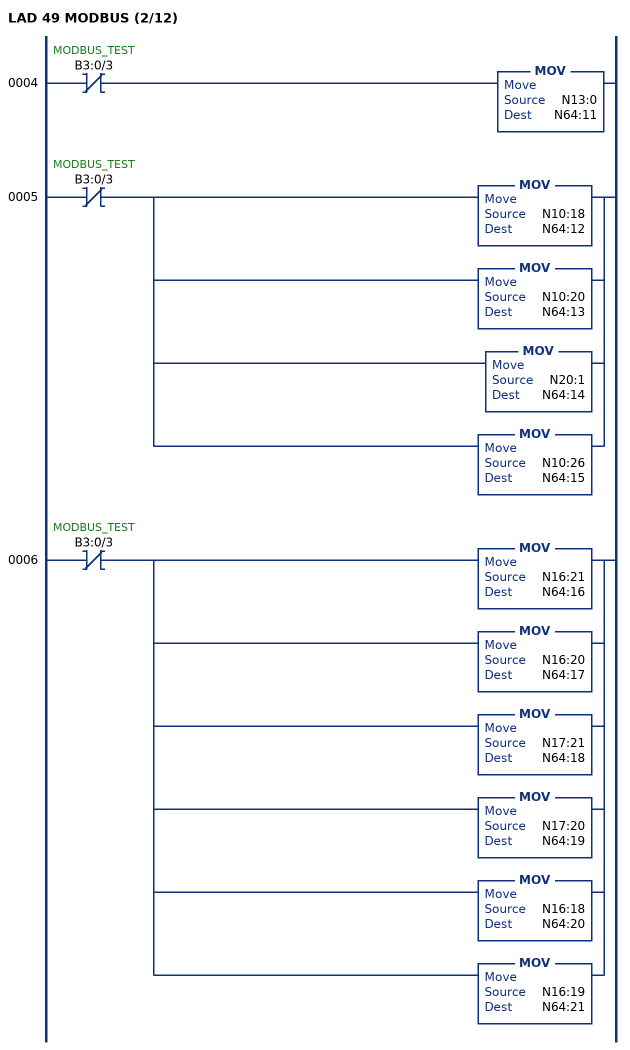
% Rung: 4 %
SOR XIO B3:0/3 MOV N13:0 N64:11 EOR
%   B3:0/3  MODBUS_TEST %
%   N13:0  REGEN_STATE  "STATE The current state of the regen process" %
% Rung: 5 %
SOR XIO B3:0/3 BST MOV N10:18 N64:12 NXB MOV N10:20 N64:13 NXB MOV N20:1 N64:14 NXB MOV N10:26 N64:15 BND EOR
%   B3:0/3  MODBUS_TEST %
%   N10:18  INLET_PX_PSIG %
%   N10:20  OUTLET_PX_PSIG %
%   N20:1  MIX_PANEL_PSIG %
%   N10:26  MFM_FLOW %
% Rung: 6 %
SOR XIO B3:0/3 BST MOV N16:21 N64:16 NXB MOV N16:20 N64:17 NXB MOV N17:21 N64:18 NXB MOV N17:20 N64:19 NXB MOV N16:18 N64:20 NXB MOV N16:19 N64:21 BND EOR
%   B3:0/3  MODBUS_TEST %
%   N16:21  ADS_A_BED_TEMP_READ %
%   N16:20  ADS_A_WALL_TEMP_READ %
%   N17:21  ADS_B_BED_TEMP_READ %
%   N17:20  ADS_B_WALL_TEMP_READ %
%   N16:18  ADS_PH_GAS_TEMP_READ %
%   N16:19  ADS_PH_ROD_TEMP_READ %

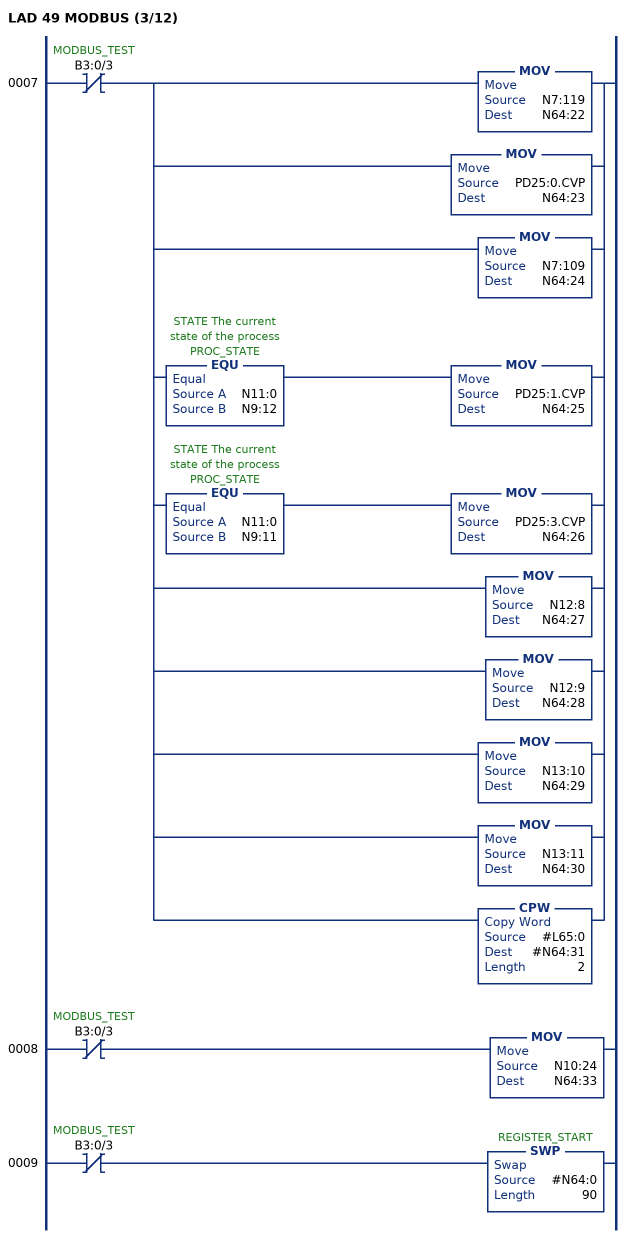
% Rung: 7 %
SOR XIO B3:0/3 BST MOV N7:119 N64:22 NXB MOV PD25:0.CVP N64:23 NXB MOV N7:109 N64:24 NXB EQU N11:0 N9:12 MOV PD25:1.CVP N64:25 NXB EQU N11:0 N9:11 MOV PD25:3.CVP N64:26 NXB MOV N12:8 N64:27 NXB MOV N12:9 N64:28 NXB MOV N13:10 N64:29 NXB MOV N13:11 N64:30 NXB CPW #L65:0 #N64:31 2 BND EOR
%   B3:0/3  MODBUS_TEST %
%   N7:119  PREHEATER_SP  "CONTROL Preheater PID Setpoint" %
%   N7:109  BLANKET_SP  "CONTROL Blanket PID Setpoint" %
%   N11:0  PROC_STATE  "STATE The current state of the process" %
%   N9:12  PROC_PURIFY_B  "STATE Process Purify B" %
%   N9:11  PROC_PURIFY_A  "STATE Process Purify A" %
%   N12:8  HRS_LEFT_IN_PURIFY %
%   N12:9  MIN_LEFT_IN_PURIFY %
%   N13:10  REGEN_HRS_LEFT  "STATUS Regen Preheater Temperature Initial Temperature" %
%   N13:11  REGEN_MIN_LEFT  "STATUS Preheater Alarm Measured temperature change" %
%   L65:0  TOTAL_FLOW %
% Rung: 8 %
SOR XIO B3:0/3 MOV N10:24 N64:33 EOR
%   B3:0/3  MODBUS_TEST %
%   N10:24  H2_SENSOR_LEVEL %
% Rung: 9 %
SOR XIO B3:0/3 SWP #N64:0 90 EOR
%   B3:0/3  MODBUS_TEST %
%   N64:0  REGISTER_START %

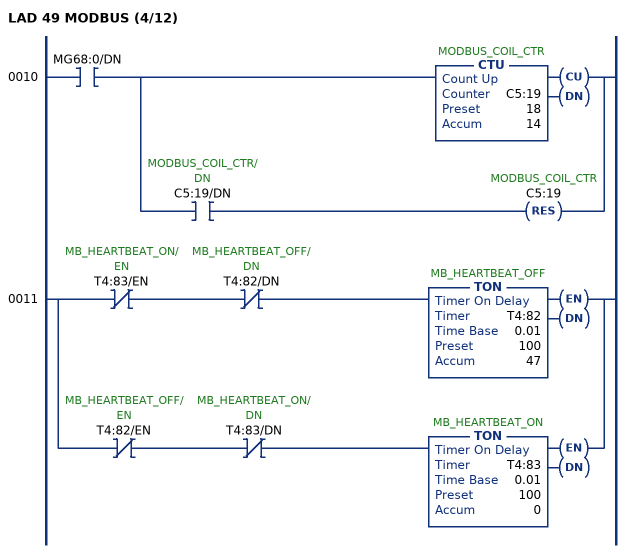
% Rung: 10 %
SOR XIC MG68:0/DN BST CTU C5:19 18 14 NXB XIC C5:19/DN RES C5:19 BND EOR
%   C5:19  MODBUS_COIL_CTR %
% Rung: 11 %
SOR BST XIO T4:83/EN XIO T4:82/DN TON T4:82 0.01 100 47 NXB XIO T4:82/EN XIO T4:83/DN TON T4:83 0.01 100 0 BND EOR
%   T4:83  MB_HEARTBEAT_ON %
%   T4:82  MB_HEARTBEAT_OFF %

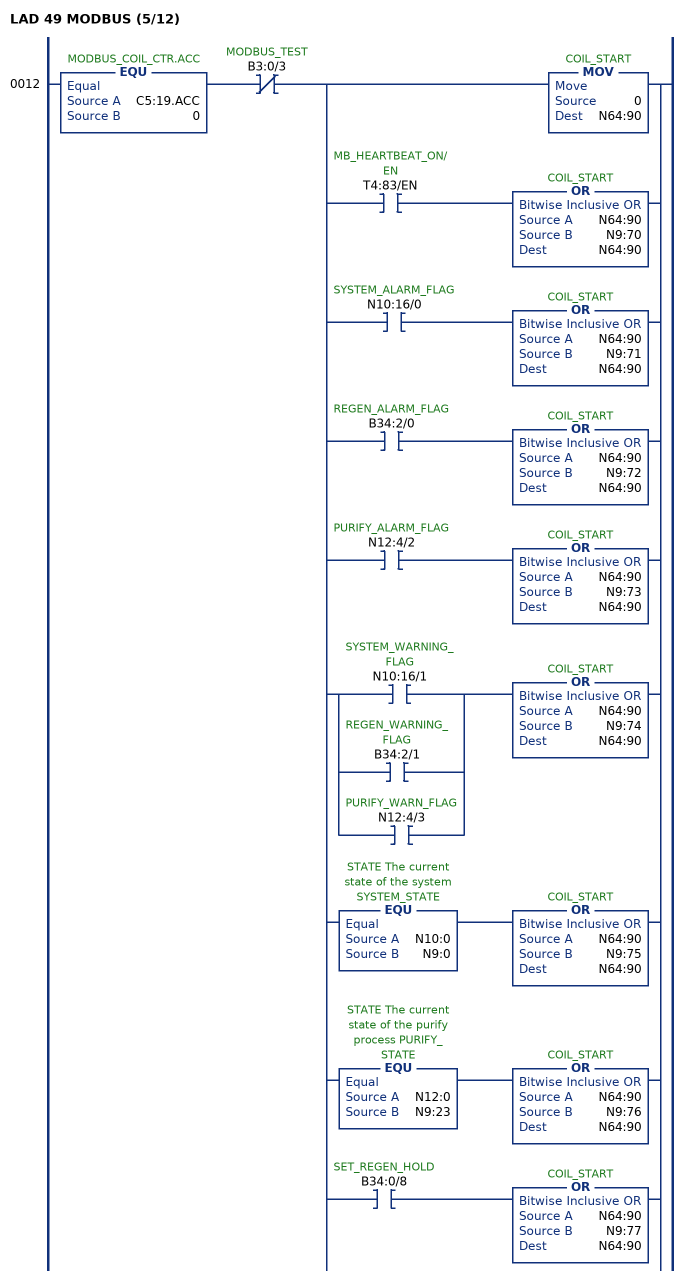

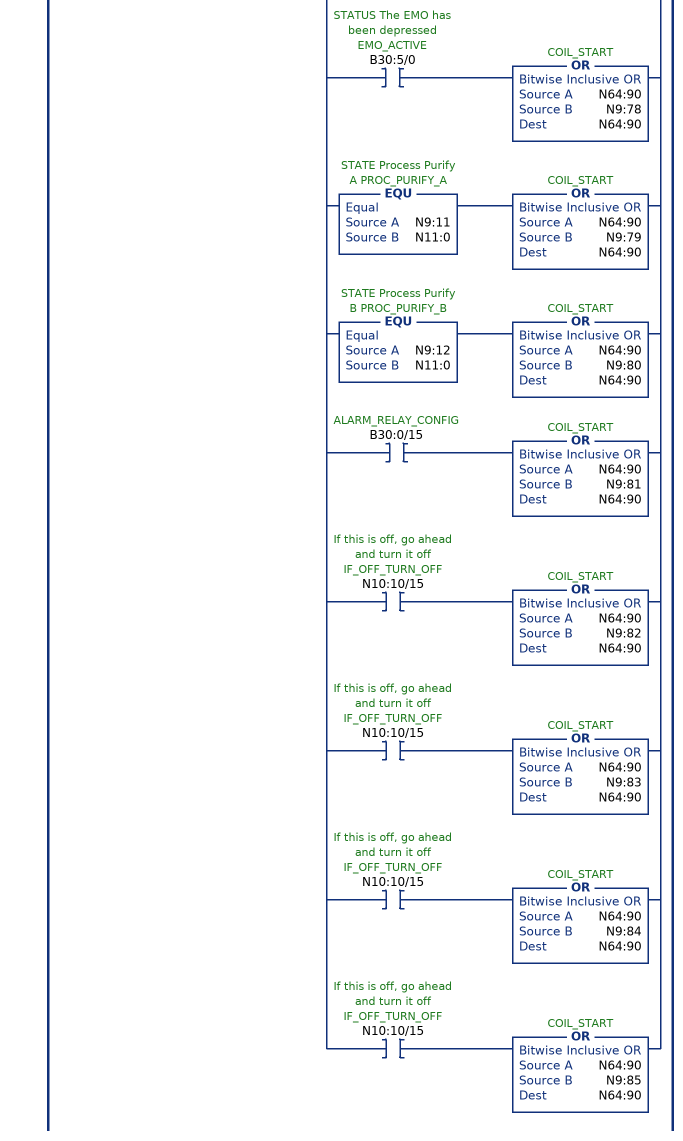
% Rung: 12 %
SOR EQU C5:19.ACC 0 XIO B3:0/3 BST MOV 0 N64:90 NXB XIC T4:83/EN OR N64:90 N9:70 N64:90 NXB XIC N10:16/0 OR N64:90 N9:71 N64:90 NXB XIC B34:2/0 OR N64:90 N9:72 N64:90 NXB XIC N12:4/2 OR N64:90 N9:73 N64:90 NXB BST XIC N10:16/1 NXB XIC B34:2/1 NXB XIC N12:4/3 BND OR N64:90 N9:74 N64:90 NXB EQU N10:0 N9:0 OR N64:90 N9:75 N64:90 NXB EQU N12:0 N9:23 OR N64:90 N9:76 N64:90 NXB XIC B34:0/8 OR N64:90 N9:77 N64:90 NXB XIC B30:5/0 OR N64:90 N9:78 N64:90 NXB EQU N9:11 N11:0 OR N64:90 N9:79 N64:90 NXB EQU N9:12 N11:0 OR N64:90 N9:80 N64:90 NXB XIC B30:0/15 OR N64:90 N9:81 N64:90 NXB XIC N10:10/15 OR N64:90 N9:82 N64:90 NXB XIC N10:10/15 OR N64:90 N9:83 N64:90 NXB XIC N10:10/15 OR N64:90 N9:84 N64:90 NXB XIC N10:10/15 OR N64:90 N9:85 N64:90 BND EOR
%   C5:19  MODBUS_COIL_CTR %
%   B3:0/3  MODBUS_TEST %
%   N64:90  COIL_START %
%   T4:83  MB_HEARTBEAT_ON %
%   N9:70  BIT_0 %
%   N10:16/0  SYSTEM_ALARM_FLAG %
%   N9:71  BIT_1 %
%   B34:2/0  REGEN_ALARM_FLAG %
%   N9:72  BIT_2 %
%   N12:4/2  PURIFY_ALARM_FLAG %
%   N9:73  BIT_3 %
%   N10:16/1  SYSTEM_WARNING_FLAG %
%   B34:2/1  REGEN_WARNING_FLAG %
%   N12:4/3  PURIFY_WARN_FLAG %
%   N9:74  BIT_4 %
%   N10:0  SYSTEM_STATE  "STATE The current state of the system" %
%   N9:0  SYSTEM_STANDBY  "STATE System Standby" %
%   N9:75  BIT_5 %
%   N12:0  PURIFY_STATE  "STATE The current state of the purify process" %
%   N9:23  PURIFY_MANUAL_HOLD  "STATE Purify Manual Hold" %
%   N9:76  BIT_6 %
%   B34:0/8  SET_REGEN_HOLD %
%   N9:77  BIT_7 %
%   B30:5/0  EMO_ACTIVE  "STATUS The EMO has been depressed" %
%   N9:78  BIT_8 %
%   N9:11  PROC_PURIFY_A  "STATE Process Purify A" %
%   N11:0  PROC_STATE  "STATE The current state of the process" %
%   N9:79  BIT_9 %
%   N9:12  PROC_PURIFY_B  "STATE Process Purify B" %
%   N9:80  BIT_10 %
%   B30:0/15  ALARM_RELAY_CONFIG %
%   N9:81  BIT_11 %
%   N10:10/15  IF_OFF_TURN_OFF  "If this is off, go ahead and turn it off" %
%   N9:82  BIT_12 %
%   N9:83  BIT_13 %
%   N9:84  BIT_14 %
%   N9:85  BIT_15 %

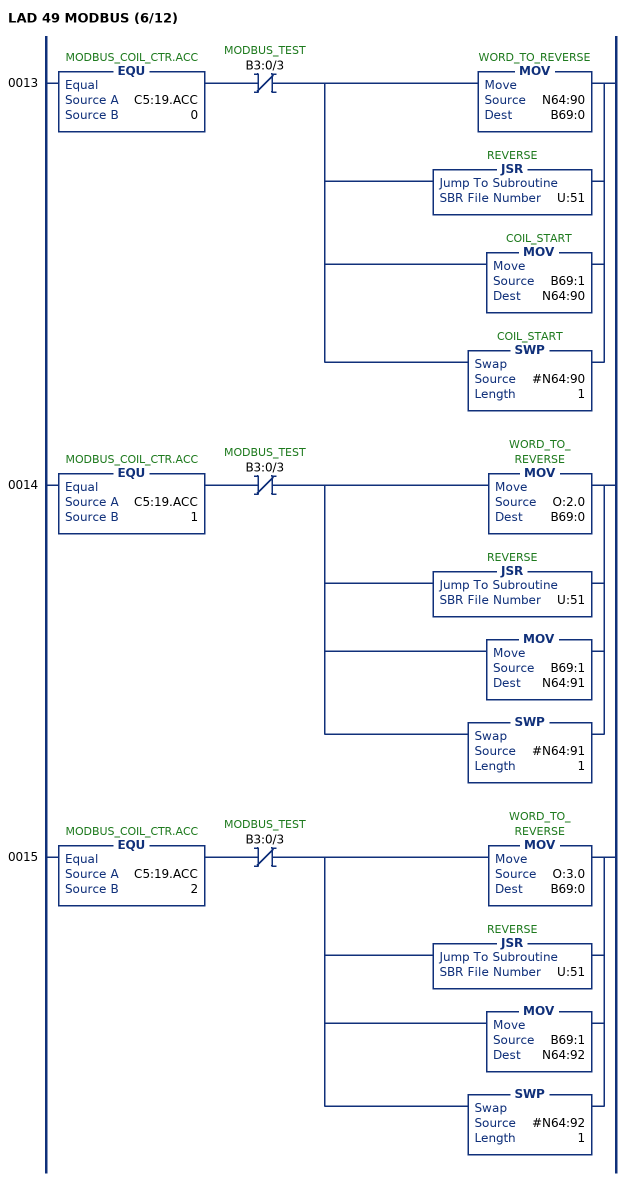
% Rung: 13 %
SOR EQU C5:19.ACC 0 XIO B3:0/3 BST MOV N64:90 B69:0 NXB JSR U:51 NXB MOV B69:1 N64:90 NXB SWP #N64:90 1 BND EOR
%   C5:19  MODBUS_COIL_CTR %
%   B3:0/3  MODBUS_TEST %
%   N64:90  COIL_START %
%   B69:0  WORD_TO_REVERSE %
%   U:51  REVERSE %
%   B69:1  REVERSED_WORD %
% Rung: 14 %
SOR EQU C5:19.ACC 1 XIO B3:0/3 BST MOV O:2.0 B69:0 NXB JSR U:51 NXB MOV B69:1 N64:91 NXB SWP #N64:91 1 BND EOR
%   C5:19  MODBUS_COIL_CTR %
%   B3:0/3  MODBUS_TEST %
%   B69:0  WORD_TO_REVERSE %
%   U:51  REVERSE %
%   B69:1  REVERSED_WORD %
% Rung: 15 %
SOR EQU C5:19.ACC 2 XIO B3:0/3 BST MOV O:3.0 B69:0 NXB JSR U:51 NXB MOV B69:1 N64:92 NXB SWP #N64:92 1 BND EOR
%   C5:19  MODBUS_COIL_CTR %
%   B3:0/3  MODBUS_TEST %
%   B69:0  WORD_TO_REVERSE %
%   U:51  REVERSE %
%   B69:1  REVERSED_WORD %

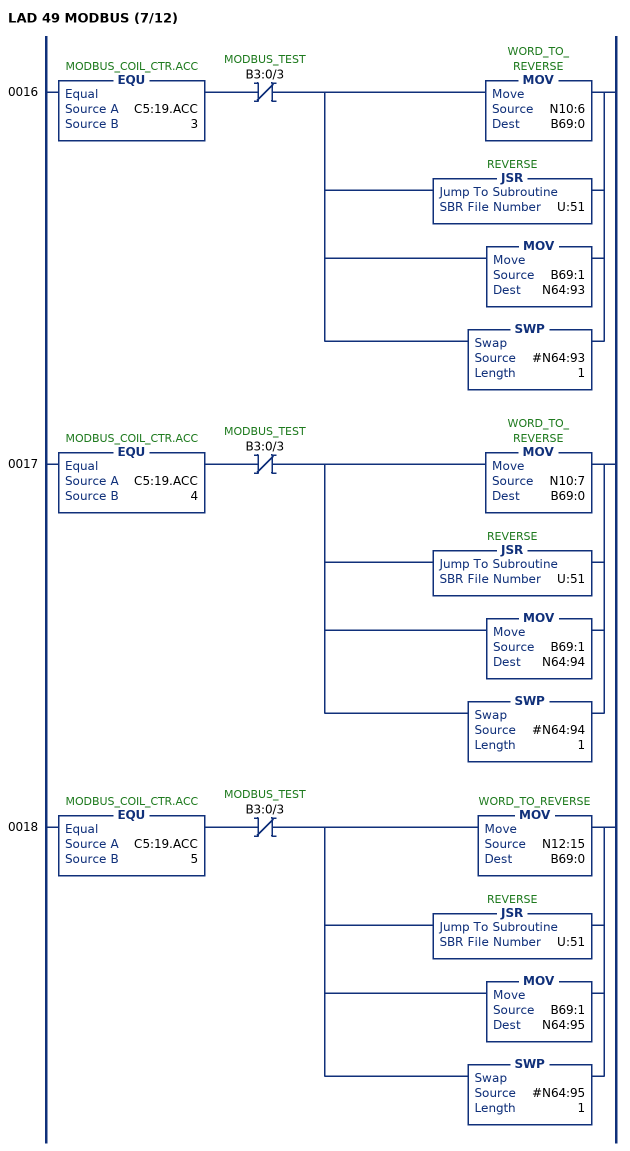
% Rung: 16 %
SOR EQU C5:19.ACC 3 XIO B3:0/3 BST MOV N10:6 B69:0 NXB JSR U:51 NXB MOV B69:1 N64:93 NXB SWP #N64:93 1 BND EOR
%   C5:19  MODBUS_COIL_CTR %
%   B3:0/3  MODBUS_TEST %
%   N10:6  SYSTEM_ALARMS_0  "ALARM System alarms" %
%   B69:0  WORD_TO_REVERSE %
%   U:51  REVERSE %
%   B69:1  REVERSED_WORD %
% Rung: 17 %
SOR EQU C5:19.ACC 4 XIO B3:0/3 BST MOV N10:7 B69:0 NXB JSR U:51 NXB MOV B69:1 N64:94 NXB SWP #N64:94 1 BND EOR
%   C5:19  MODBUS_COIL_CTR %
%   B3:0/3  MODBUS_TEST %
%   N10:7  SYSTEM_ALARMS_1  "ALARM System alarms" %
%   B69:0  WORD_TO_REVERSE %
%   U:51  REVERSE %
%   B69:1  REVERSED_WORD %
% Rung: 18 %
SOR EQU C5:19.ACC 5 XIO B3:0/3 BST MOV N12:15 B69:0 NXB JSR U:51 NXB MOV B69:1 N64:95 NXB SWP #N64:95 1 BND EOR
%   C5:19  MODBUS_COIL_CTR %
%   B3:0/3  MODBUS_TEST %
%   N12:15  PURIFY_ALARMS_0 %
%   B69:0  WORD_TO_REVERSE %
%   U:51  REVERSE %
%   B69:1  REVERSED_WORD %

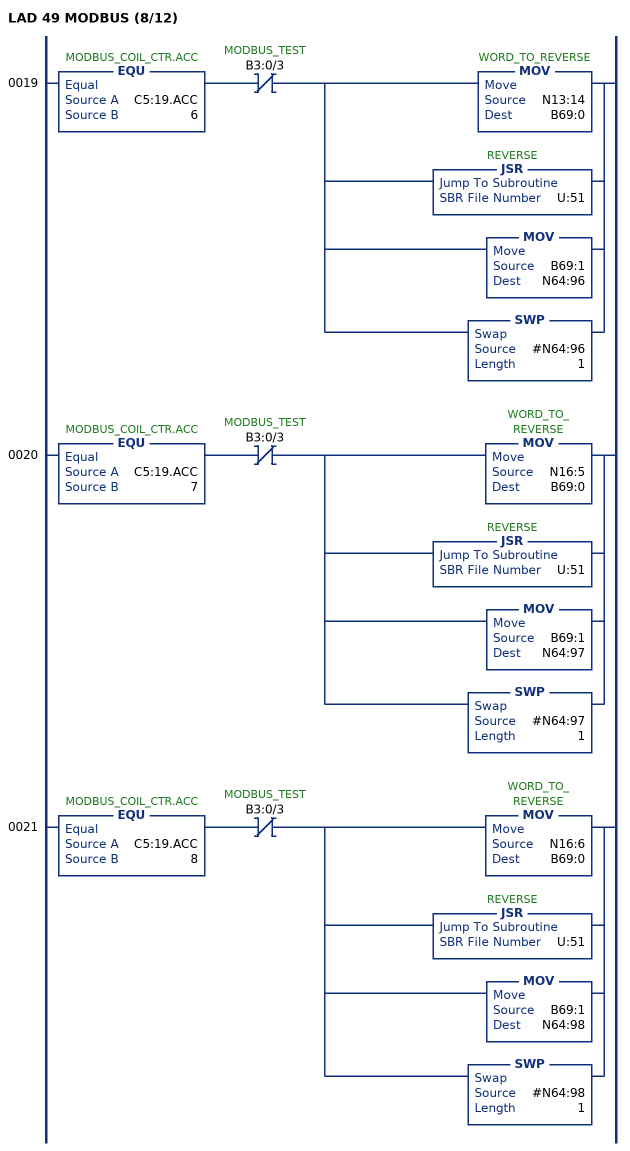
% Rung: 19 %
SOR EQU C5:19.ACC 6 XIO B3:0/3 BST MOV N13:14 B69:0 NXB JSR U:51 NXB MOV B69:1 N64:96 NXB SWP #N64:96 1 BND EOR
%   C5:19  MODBUS_COIL_CTR %
%   B3:0/3  MODBUS_TEST %
%   N13:14  REGEN_ALARMS_0 %
%   B69:0  WORD_TO_REVERSE %
%   U:51  REVERSE %
%   B69:1  REVERSED_WORD %
% Rung: 20 %
SOR EQU C5:19.ACC 7 XIO B3:0/3 BST MOV N16:5 B69:0 NXB JSR U:51 NXB MOV B69:1 N64:97 NXB SWP #N64:97 1 BND EOR
%   C5:19  MODBUS_COIL_CTR %
%   B3:0/3  MODBUS_TEST %
%   N16:5  ADS_A_ALARMS_0  "ALARM ADS A Alarms" %
%   B69:0  WORD_TO_REVERSE %
%   U:51  REVERSE %
%   B69:1  REVERSED_WORD %
% Rung: 21 %
SOR EQU C5:19.ACC 8 XIO B3:0/3 BST MOV N16:6 B69:0 NXB JSR U:51 NXB MOV B69:1 N64:98 NXB SWP #N64:98 1 BND EOR
%   C5:19  MODBUS_COIL_CTR %
%   B3:0/3  MODBUS_TEST %
%   N16:6  ADS_A_ALARMS_1  "ALARM ADS A Alarms" %
%   B69:0  WORD_TO_REVERSE %
%   U:51  REVERSE %
%   B69:1  REVERSED_WORD %

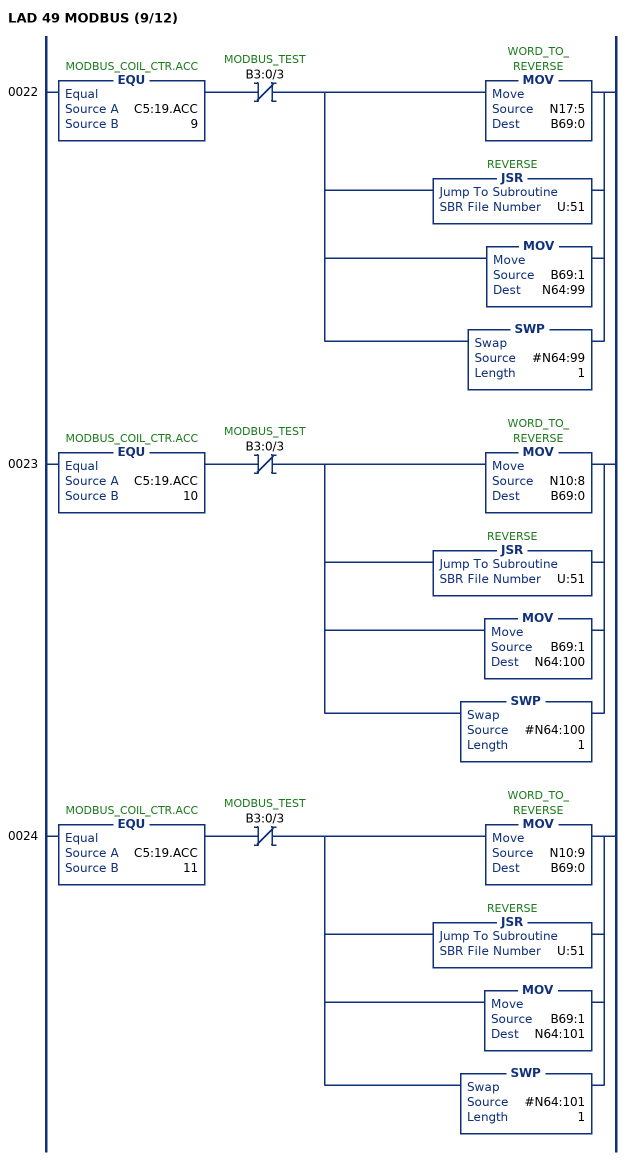
% Rung: 22 %
SOR EQU C5:19.ACC 9 XIO B3:0/3 BST MOV N17:5 B69:0 NXB JSR U:51 NXB MOV B69:1 N64:99 NXB SWP #N64:99 1 BND EOR
%   C5:19  MODBUS_COIL_CTR %
%   B3:0/3  MODBUS_TEST %
%   N17:5  ADS_B_ALARMS_0  "ALARM Alarm bits" %
%   B69:0  WORD_TO_REVERSE %
%   U:51  REVERSE %
%   B69:1  REVERSED_WORD %
% Rung: 23 %
SOR EQU C5:19.ACC 10 XIO B3:0/3 BST MOV N10:8 B69:0 NXB JSR U:51 NXB MOV B69:1 N64:100 NXB SWP #N64:100 1 BND EOR
%   C5:19  MODBUS_COIL_CTR %
%   B3:0/3  MODBUS_TEST %
%   N10:8  SYSTEM_WARNINGS_0  "WARNING System Warnings" %
%   B69:0  WORD_TO_REVERSE %
%   U:51  REVERSE %
%   B69:1  REVERSED_WORD %
% Rung: 24 %
SOR EQU C5:19.ACC 11 XIO B3:0/3 BST MOV N10:9 B69:0 NXB JSR U:51 NXB MOV B69:1 N64:101 NXB SWP #N64:101 1 BND EOR
%   C5:19  MODBUS_COIL_CTR %
%   B3:0/3  MODBUS_TEST %
%   N10:9  SYSTEM_WARNINGS_1  "WARNING System Warnings" %
%   B69:0  WORD_TO_REVERSE %
%   U:51  REVERSE %
%   B69:1  REVERSED_WORD %

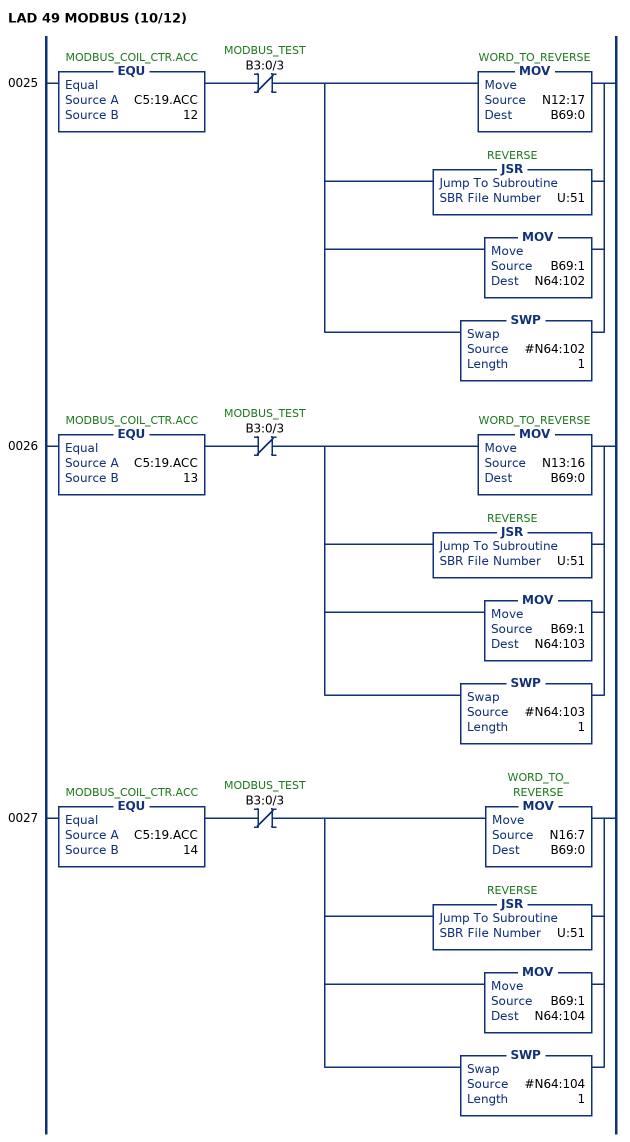
% Rung: 25 %
SOR EQU C5:19.ACC 12 XIO B3:0/3 BST MOV N12:17 B69:0 NXB JSR U:51 NXB MOV B69:1 N64:102 NXB SWP #N64:102 1 BND EOR
%   C5:19  MODBUS_COIL_CTR %
%   B3:0/3  MODBUS_TEST %
%   N12:17  PURIFY_WARNINGS_0 %
%   B69:0  WORD_TO_REVERSE %
%   U:51  REVERSE %
%   B69:1  REVERSED_WORD %
% Rung: 26 %
SOR EQU C5:19.ACC 13 XIO B3:0/3 BST MOV N13:16 B69:0 NXB JSR U:51 NXB MOV B69:1 N64:103 NXB SWP #N64:103 1 BND EOR
%   C5:19  MODBUS_COIL_CTR %
%   B3:0/3  MODBUS_TEST %
%   N13:16  REGEN_WARNINGS_0 %
%   B69:0  WORD_TO_REVERSE %
%   U:51  REVERSE %
%   B69:1  REVERSED_WORD %
% Rung: 27 %
SOR EQU C5:19.ACC 14 XIO B3:0/3 BST MOV N16:7 B69:0 NXB JSR U:51 NXB MOV B69:1 N64:104 NXB SWP #N64:104 1 BND EOR
%   C5:19  MODBUS_COIL_CTR %
%   B3:0/3  MODBUS_TEST %
%   N16:7  ADS_A_WARNINGS_0  "WARNING ADS A Warnings" %
%   B69:0  WORD_TO_REVERSE %
%   U:51  REVERSE %
%   B69:1  REVERSED_WORD %

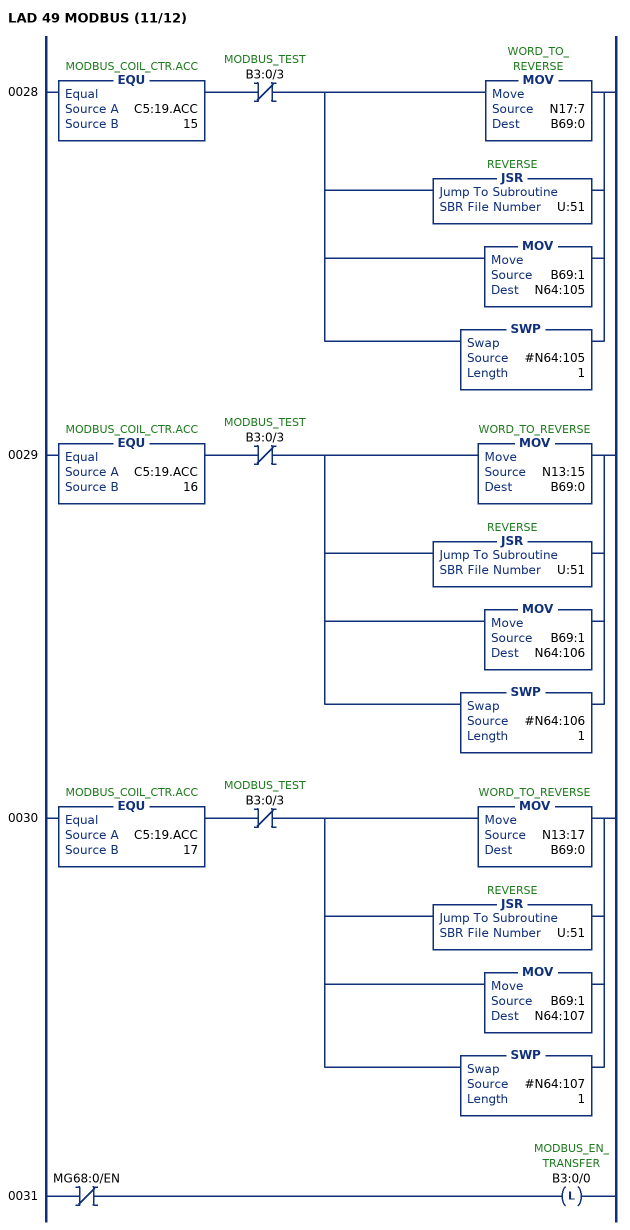
% Rung: 28 %
SOR EQU C5:19.ACC 15 XIO B3:0/3 BST MOV N17:7 B69:0 NXB JSR U:51 NXB MOV B69:1 N64:105 NXB SWP #N64:105 1 BND EOR
%   C5:19  MODBUS_COIL_CTR %
%   B3:0/3  MODBUS_TEST %
%   N17:7  ADS_B_WARNINGS_0  "WARNING Warning bits" %
%   B69:0  WORD_TO_REVERSE %
%   U:51  REVERSE %
%   B69:1  REVERSED_WORD %
% Rung: 29 %
SOR EQU C5:19.ACC 16 XIO B3:0/3 BST MOV N13:15 B69:0 NXB JSR U:51 NXB MOV B69:1 N64:106 NXB SWP #N64:106 1 BND EOR
%   C5:19  MODBUS_COIL_CTR %
%   B3:0/3  MODBUS_TEST %
%   N13:15  REGEN_ALARMS_1 %
%   B69:0  WORD_TO_REVERSE %
%   U:51  REVERSE %
%   B69:1  REVERSED_WORD %
% Rung: 30 %
SOR EQU C5:19.ACC 17 XIO B3:0/3 BST MOV N13:17 B69:0 NXB JSR U:51 NXB MOV B69:1 N64:107 NXB SWP #N64:107 1 BND EOR
%   C5:19  MODBUS_COIL_CTR %
%   B3:0/3  MODBUS_TEST %
%   N13:17  REGEN_WARNINGS_1 %
%   B69:0  WORD_TO_REVERSE %
%   U:51  REVERSE %
%   B69:1  REVERSED_WORD %
% Rung: 31 %
SOR XIO MG68:0/EN OTL B3:0/0 EOR
%   B3:0/0  MODBUS_EN_TRANSFER %

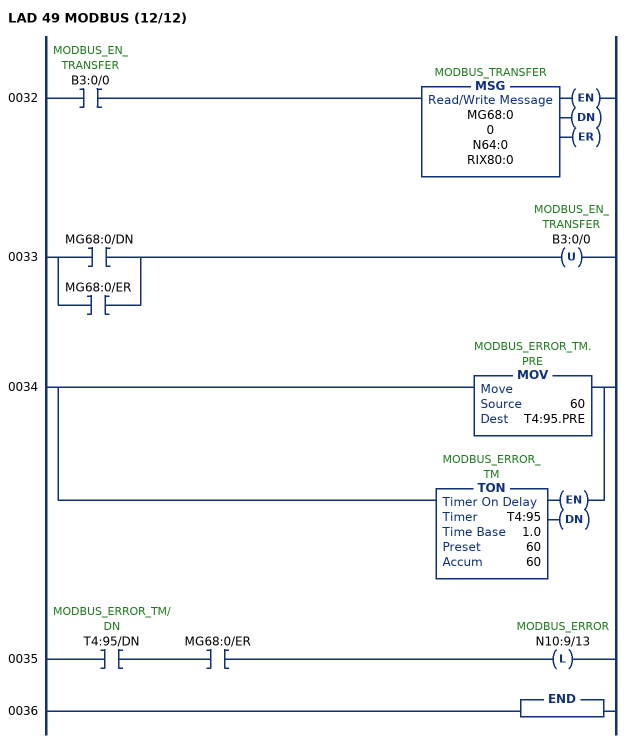
% Rung: 32 %
SOR XIC B3:0/0 MSG MG68:0 0 N64:0 RIX80:0 EOR
%   B3:0/0  MODBUS_EN_TRANSFER %
%   MSG set-up: CIP Generic | 33 | 0 | ? | 0 | 0 | 0 | 0 | 172.16.14.73:502 | 0 | 0 | 172.16.14.73 | RIX80:0 | 10 | 4 | 150 | 3 | 4 | 96 | 3 | 252 | N64:0 %
%   MG68:0  MODBUS_TRANSFER %
%   N64:0  REGISTER_START %
% Rung: 33 %
SOR BST XIC MG68:0/DN NXB XIC MG68:0/ER BND OTU B3:0/0 EOR
%   B3:0/0  MODBUS_EN_TRANSFER %
% Rung: 34 %
SOR BST MOV 60 T4:95.PRE NXB TON T4:95 1.0 60 60 BND EOR
%   T4:95  MODBUS_ERROR_TM %
% Rung: 35 %
SOR XIC T4:95/DN XIC MG68:0/ER OTL N10:9/13 EOR
%   T4:95  MODBUS_ERROR_TM %
%   N10:9/13  MODBUS_ERROR %
% Rung: 36 %
SOR END EOR

LADDER 50 "PLC_FAULT"
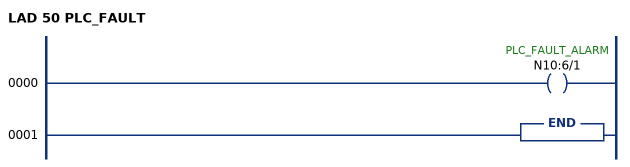
% Rung: 0 %
SOR OTE N10:6/1 EOR
%   N10:6/1  PLC_FAULT_ALARM %
% Rung: 1 %
SOR END EOR

LADDER 51 "REVERSE"
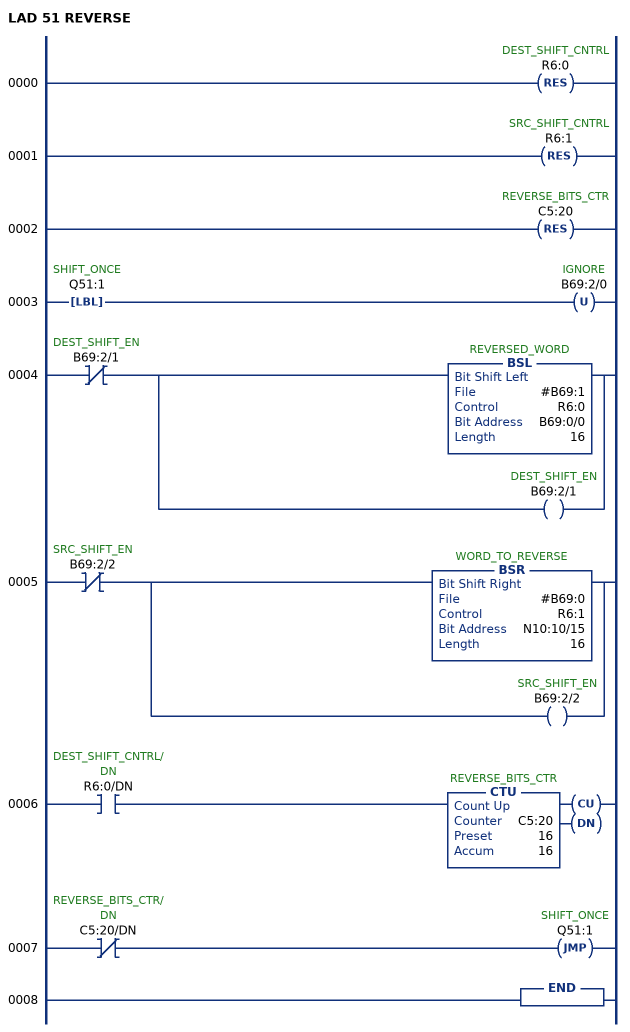
% Rung: 0 %
SOR RES R6:0 EOR
%   R6:0  DEST_SHIFT_CNTRL %
% Rung: 1 %
SOR RES R6:1 EOR
%   R6:1  SRC_SHIFT_CNTRL %
% Rung: 2 %
SOR RES C5:20 EOR
%   C5:20  REVERSE_BITS_CTR %
% Rung: 3 %
SOR LBL Q51:1 OTU B69:2/0 EOR
%   Q51:1  SHIFT_ONCE %
%   B69:2/0  IGNORE %
% Rung: 4 %
SOR XIO B69:2/1 BST BSL #B69:1 R6:0 B69:0/0 16 NXB OTE B69:2/1 BND EOR
%   B69:2/1  DEST_SHIFT_EN %
%   B69:1  REVERSED_WORD %
%   R6:0  DEST_SHIFT_CNTRL %
% Rung: 5 %
SOR XIO B69:2/2 BST BSR #B69:0 R6:1 N10:10/15 16 NXB OTE B69:2/2 BND EOR
%   B69:2/2  SRC_SHIFT_EN %
%   B69:0  WORD_TO_REVERSE %
%   R6:1  SRC_SHIFT_CNTRL %
%   N10:10/15  IF_OFF_TURN_OFF  "If this is off, go ahead and turn it off" %
% Rung: 6 %
SOR XIC R6:0/DN CTU C5:20 16 16 EOR
%   R6:0  DEST_SHIFT_CNTRL %
%   C5:20  REVERSE_BITS_CTR %
% Rung: 7 %
SOR XIO C5:20/DN JMP Q51:1 EOR
%   C5:20  REVERSE_BITS_CTR %
%   Q51:1  SHIFT_ONCE %
% Rung: 8 %
SOR END EOR

OTHER DOCUMENTED ADDRESSES
  B26:2/2  H2_LEAK_ALM_EN
  B30:0  CONFIG_BITS_HARDWARE  "CONFIG Hardware options installed"
  B30:1/0  MOIST_SENS_ALM
  B30:5  SYSTEM_STATUS_0  "STATUS System Status of system contro entities"
  B30:5/6  LP_REGEN_PS6_TRIPPED
  B31:2  SYSTEM_HMI_CMD_0  "COMMAND HMI Commands"
  B31:3  SYSTEM_HMI_CMD_1  "COMMAND HMI Commands"
  B31:4  SYSTEM_HMI_CMD_2  "COMMAND HMI Commands"
  B31:5  SYSTEM_HMI_CMD_3
  B31:6  SYSTEM_HMI_CMD_4  "COMMAND HMI Commands"
  B31:7  SYSTEM_HMI_CMD_5  "COMMAND HMI Commands"
  B33:0  PURIFY_HMI_CMDS
  B33:0/1  DEF_PURIFY_MAX
  B33:1/0  PUR_EQUATION_1_FLAG
  B33:1/1  PUR_EQUATION_2_FLAG
  B33:1/2  PURIFY_DEF_FLAG
  B33:1/3  PURIFY_DEF_ONE_SHOT
  B34:0  REGEN_HMI_CMDS
  B34:2  REGEN_FLAGS
  B35:2  MANUAL_HMI_CMNDS_0
  B36:1/2  PURGE_COMPLETE
  DFILE:0  "OUTPUT"
  DFILE:1  "INPUT"
  DFILE:2  "STATUS"
  DFILE:3  "BINARY"
  DFILE:4  "TIMER"
  DFILE:5  "COUNTER"
  DFILE:6  "CONTROL"
  DFILE:7  "SYSTEM CFG Maintains the values that characterize t he system"
  DFILE:8  "FLOAT"
  DFILE:9  "CONSTANTS The collection of sy stem and subsystem c onstants"
  DFILE:10  "SYSTEM Contain the values f or system control"
  DFILE:11  "PROCESS Contains the values for the processing m achine"
  DFILE:12  "PURIFY Contains the values required for purify"
  DFILE:13  "REGEN Contains the values required for regen"
  DFILE:15  "MANUAL CTL Contains the data fo r the manual valve c ontrol"
  DFILE:16  "ADSORBER_A Contains the values for Adsorber A"
  DFILE:17  "ADSORBER_B Contains the values required for Adsorbe r B"
  DFILE:19  "BYPASS"
  DFILE:20  "MIX PANEL"
  DFILE:21  "OUTLET"
  DFILE:25  "PID HEATER"
  DFILE:30  "SYSTEM CFG"
  DFILE:31  "SYSTEM"
  DFILE:32  "PROCESS"
  DFILE:33  "PURIFY"
  DFILE:34  "REGEN"
  DFILE:35  "MANUAL CTL"
  DFILE:36  "ADSORBER_A"
  DFILE:37  "ADSORBER_B"
  DFILE:38  "BYPASS"
  DFILE:52  "SERIAL"
  DFILE:64  "MODBUS"
  DFILE:65  "TOTAL FLOW"
  F206:0  PFY_TIME_MIN_ALLOWED
  L202:0  HMI_STS_GETTER
  MS1_ISNTALLED  
  N7:0  CONFIG_BIT_ALM
  N7:1  CONFIG_BITS_ALM_O  "CONFIG System alarms enable"
  N7:2  CONFIG_BITS_ALM_1  "CONFIG System alarms enable"
  N7:2/3  MOIST_SENS_ALM_EN
  N7:3  CONFIG_BITS_WARN_0  "CONFIG System warnings enable"
  N7:4  CONFIG_BITS_WARN_1  "CONFIG System warnings enable"
  N7:5  CONFIG_BIT_WARN
  N7:6  CONFIG_OPEN_TC_ALM
  N7:7  CONFIG_OPEN_TC_WARN
  N7:8  MOIST_SENS_ALM_SETP
  N9:15  PROC_REGEN_C  "STATE Process Regen C"
  N9:16  PROC_REGEN_D  "STATE Process Regen D"
  N10:10  SYSTEM_CONTROL  "CONTROL System Bits used to manipulate hardware"
  N10:10/0  ADS_PH_TPO  "CONTROL ADS PH Time proportioned output"
  N10:10/1  ADS_BLANKET_TPO  "CONTROL ADS Blanket Time proportioned output"
  N10:16  SYSTEM_FLAGS_1
  N12:4  PURIFY_FLAGS_0  "STATUS Flags used by the purify process"
  N12:5  PURIFY_CONTROL  "CONTROL Control bits used by the purify process to change hardware states"
  N12:10  PURIFY_FACTOR  "CONFIG The percent output requested by the operator (percent)"
  N12:12  PURIFY_CALC_0  "CONFIG Math result placeholder for the purify time calculation"
  N12:13  PURIFY_FACTOR_TIME
  N13:5  REGEN_CONTROL  "CONTROL Regen Bits used to manipulate hardware"
  N15:4  MANUAL_FLAGS_0
  N16:3  ADS_A_FLAGS_0  "STATUS Flags used for Adsorber A"
  N17:3  ADS_B_FLAGS_0  "STATUS Flags used for Adsorber B"
  N19:1  BYPASS_COMMAND  "HMI Commands received from the HMI"
  N207:3  PURIFY_MAX_FLOW_RATE
  N207:6  PURIFY_TIME_RESULT
  O:0.0/5  BUZZER_OUT  "Alarm Buzzer Control"
  T4:48  MOIST_SENS_ALM_TMR
  T4:96  LOW_PLC_BATT_WRN_TMR  "Low PLC battery warning timer."

COMMENTS NOT ATTACHED TO A CURRENT RUNG
  B58:0/0: UPS Failure Defaults
  N7:3/6: SYSTEM DEFAULTS / Purify High Temperature Defaults
  B31:4/11: Gas Type Selection
  N7:8: Scale analog inputs / TODO: Do we need to add the ability to adjust the ammonia sensor scaling?
  N7:2/9: Regen Preheater High Temp Rod Defaults
  N7:7/7: Open Thermocouple Defaults
  N12:14: Purify Max Time Default
  N12:10: PURIFY DEFAULTS / Purify Defaults
  N7:119: Regen Adsorber Preheater PID and Limits Defaults
  N7:109: Regen Adsorber Blanket PID and Limits Defaults
  N7:4/13: Blend Gas Leak Defaults
  C66:0.PRE: Regen Equalize Time Default
  N10:6/9: SYSTEM ALARMS AND WARNINGS / Low PLC Battery Alarm and Warning
  T4:26: Main Power Fail Alarm and Warning
  T4:28: Control Power Fail Alarm and Warning
  T62:0: SCREEN COMMS / Screen Comms Alarm
  T4:38: External Pneumatic Low Pressure Alarm
  N13:16/10: INTERNAL PNEUMATIC LOW PRESSURE / Internal Pneumatic Low Pressure Alarm and Warning
  B34:2/1: Regen Warning Flag
  N13:8: Preheater PID and Limits Defaults
  B54:0/0: UPS Fault
  N207:5: 3 = SWAPPING BEDS
  N7:0/1: Flame Detector Defaults
  N10:5/0: IR Flame Detector

REVISION NOTES
  0: moved some bits out of N7 into B30
  1: moved bits out of N10 into B31
  2: moved bits from N15 into B35
  3: added the final data files. didn't need to move any bits
  4: updated configuration for TC and AI cards. updated DO module point assignments
  5: added logic for double-acting purify valves
  6: added rod and blanket limits
  7: added tags for default buttons
  8: cleaning up bed b pid control code
  9: removed h2 sensor and moved moisture sensor to channel 6
  10: changed processor name
  11: added px3 reading
  12: added call to mix panel routine
  13: test ok
  14: trying to clear plc fault by entering new pid default parameters
  15: changed stored PID values so that it maybe doesn't fault the PLC
  16: copid in new PID values from PS21
  17: cleared out the data table
  18: changed ADS_TC_OPEN_SP to 13700 by default
  19: setting default PID parameters
  20: added in preheater and blanket setpoints
  21: lots of changes to PID control
  22: fixed up PID defaults
  23: done testing
  24: got rid of separate PID defaults
  25: fixed loop update time bug in preheater defaults
  26: PID control done
  27: ok, now it's done. made Adsorber B use the same PID parameters as Adsorber A.
  28: added control for AV11 to system routine
  29: moved mixing panel valves into mixing panel routine
  30: some small fixes to the processing subroutine.
  31: cleaned up manual valve control for AV10, 11
  32: minor edit to purify factor calculation
  33: made some fixes to ADS_A routine including adding another state buffer for adsorber-only alarms.
  34: fixed up ADS_B routine so that it's like ADS_B
  35: Regen sequence modified and default regen paramters added
  36: added regen default comments
  37: added regen steps to constants
  38: Regen counter condition resets added
  39: Fixed regen standby buffer
  40: Regen buffering and sequencing checked and fixed
  41: Merged
  42: remove alarm aknowledge
  43: Updated alarm tag names
  44: PH fault changed
  45: manual mode PID taop PID control
  46: Added fail to cool alarm and warning
  47: trying to fix ph fault
  48: fixing open tc
  49: fixed open tc logic
  50: ok, now it's fixed

DATA TABLE (non-zero values as saved)
DATA T4
% .PRE .ACC %
% T4:0 % 6 0
% T4:1 % 60 0
% T4:2 % 6 0
% T4:3 % 120 0
% T4:4 % 60 0
% T4:5 % 60 0
% T4:6 % 1000 0
% T4:7 % 1000 0
% T4:8 % 5 0
% T4:9 % 5 0
% T4:10 % 5 0
% T4:11 % 5 0
% T4:12 % 5 0
% T4:13 % 5 0
% T4:14 % 5 0
% T4:15 % 5 0
% T4:16 % 21600 0
% T4:17 % 21600 0
% T4:18 % 21600 0
% T4:19 % 21600 0
% T4:20 % 5 0
% T4:21 % 5 0
% T4:22 % 5 0
% T4:23 % 5 0
% T4:24 % 5 0
% T4:25 % 5 0
% T4:26 % 30 0
% T4:27 % 30 0
% T4:28 % 5 0
% T4:29 % 5 0
% T4:30 % 60 0
% T4:31 % 60 0
% T4:32 % 5 0
% T4:33 % 5 0
% T4:34 % 5 0
% T4:35 % 5 0
% T4:36 % 5 0
% T4:37 % 5 0
% T4:38 % 5 0
% T4:39 % 60 0
% T4:40 % 5 0
% T4:41 % 5 0
% T4:42 % 5 0
% T4:43 % 5 0
% T4:44 % 5 5
% T4:45 % 60 0
% T4:46 % 500 76
% T4:47 % 60 46
% T4:48 % 5 0
% T4:49 % 5 0
% T4:50 % 180 0
% T4:51 % 5 0
% T4:52 % 5 0
% T4:53 % 5 0
% T4:54 % 120 0
% T4:55 % 60 0
% T4:56 % 60 0
% T4:57 % 30 0
% T4:58 % 30 0
% T4:59 % 60 0
% T4:60 % 60 0
% T4:61 % 10 0
% T4:62 % 10 0
% T4:63 % 60 0
% T4:64 % 60 0
% T4:65 % 60 0
% T4:66 % 60 0
% T4:67 % 60 0
% T4:68 % 60 0
% T4:69 % 60 0
% T4:70 % 5 0
% T4:71 % 5 0
% T4:72 % 5 0
% T4:73 % 5 0
% T4:74 % 60 0
% T4:75 % 60 0
% T4:76 % 5 0
% T4:77 % 5 0
% T4:78 % 5 0
% T4:79 % 5 0
% T4:80 % 5 0
% T4:81 % 5 0
% T4:82 % 100 47
% T4:83 % 100 0
% T4:84 % 5 0
% T4:85 % 5 0
% T4:86 % 5 0
% T4:87 % 5 0
% T4:88 % 1 0
% T4:89 % 500 0
% T4:90 % 5 0
% T4:91 % 5 0
% T4:92 % 60 0
% T4:93 % 5 0
% T4:94 % 90 0
% T4:95 % 60 60
% T4:97 % 5 0
% T4:98 % 5 0
% T4:99 % 5 0
% T4:100 % 5 0
% T4:101 % 5 0
% T4:102 % 5 0
% T4:103 % 5 0
% T4:104 % 5 0
% T4:105 % 5 0
% T4:106 % 5 0
% T4:107 % 5 0
% T4:108 % 5 0
% T4:109 % 5 0
% T4:110 % 5 0
% T4:111 % 5 0
DATA C5
% .PRE .ACC %
% C5:0 % 120 0
% C5:1 % 60 31
% C5:2 % 24 8
% C5:3 % 32767 6
% C5:4 % 240 0
% C5:5 % 180 25
% C5:6 % 30 0
% C5:7 % 12 0
% C5:8 % 480 0
% C5:9 % 5 0
% C5:10 % 5 0
% C5:11 % 5 0
% C5:12 % 5 0
% C5:13 % 30 0
% C5:14 % 12 0
% C5:15 % 15 0
% C5:16 % 8 0
% C5:17 % 720 0
% C5:18 % 720 0
% C5:19 % 18 14
% C5:20 % 16 16
DATA R6
% .LEN .POS %
% R6:0 % 16 0
% R6:1 % 16 0
DATA N64
% N64:0 % 28684 0 0 0 0 0 0 0 0 0
